// One diagnostic entry.
TYPE DebugStruct :
STRUCT
	iSource: I_Debug; // Object that reported the message.
	sComment: Str; // Diagnostic text.
END_STRUCT
END_TYPE

(* stored: Version 1.1.0.1
   DUT DebugStruct: Id {ff4f564d-74f0-4be1-895f-bc1505d9c37a} *)
